// Tests exercise the public input/output and command contracts.
FUNCTION_BLOCK FB_DigitalInput_Test EXTENDS TcUnit.FB_TestSuite

InitialStateClean();
RawSignalPassthroughWithNoDebounce();
InvertFlipsDebouncedValueNotRaw();
RisingEdgePulseOneScan();
FallingEdgePulseOneScan();
DebounceOnBlocksRisingEdgeUntilElapsed();
DebounceOffHoldsSignalHighAfterRawGoesLow();
BadQualityHoldsLastRawValue();
QualityTagSurfacesInStatus();
ClampedQualityReadsAsGood();

METHOD InitialStateClean
VAR
    fb : TcForge.FB_DigitalInput;
END_VAR
TEST('InitialStateClean');

fb(inpQuality := TcForge.E_IO_Quality.GOOD);

AssertFalse(
    Condition := fb.sts.value,
    Message   := 'Fresh instance must read LOW when the physical input is LOW');
AssertFalse(
    Condition := fb.sts.rawValue,
    Message   := 'Fresh instance must report the raw input LOW');
AssertFalse(
    Condition := fb.sts.risingEdge,
    Message   := 'Fresh instance must not emit a spurious rising edge');
AssertFalse(
    Condition := fb.sts.fallingEdge,
    Message   := 'Fresh instance must not emit a spurious falling edge');
AssertFalse(
    Condition := fb.sts.header.faulted,
    Message   := 'Fresh instance must not be faulted');

TEST_FINISHED();
END_METHOD

METHOD RawSignalPassthroughWithNoDebounce
VAR
    fb : TcForge.FB_DigitalInput;
END_VAR
TEST('RawSignalPassthroughWithNoDebounce');

// Default cfg: no debounce, no invert. Raw hardware bit flushes through
// to value in one cycle.
fb.inSignal := TRUE;
fb(inpQuality := TcForge.E_IO_Quality.GOOD);

AssertTrue(
    Condition := fb.sts.rawValue,
    Message   := 'rawValue must echo the hardware bit under GOOD quality');
AssertTrue(
    Condition := fb.sts.value,
    Message   := 'With no debounce and no invert the conditioned value must match the raw bit');

TEST_FINISHED();
END_METHOD

METHOD InvertFlipsDebouncedValueNotRaw
VAR
    fb : TcForge.FB_DigitalInput;
END_VAR
TEST('InvertFlipsDebouncedValueNotRaw');

// Invert must apply to the debounced / published value but the raw
// reading should stay true-to-the-wire so troubleshooters can see what
// the hardware is actually doing.
fb.cfg.invert := TRUE;
fb.inSignal := TRUE;
fb(inpQuality := TcForge.E_IO_Quality.GOOD);

AssertTrue(
    Condition := fb.sts.rawValue,
    Message   := 'rawValue must echo the wire value independent of invert');
AssertFalse(
    Condition := fb.sts.value,
    Message   := 'invert must flip the conditioned value (active-low sensor semantics)');

TEST_FINISHED();
END_METHOD

METHOD RisingEdgePulseOneScan
VAR
    fb : TcForge.FB_DigitalInput;
END_VAR
TEST('RisingEdgePulseOneScan');

fb.inSignal := FALSE;
fb(inpQuality := TcForge.E_IO_Quality.GOOD);

fb.inSignal := TRUE;
fb(inpQuality := TcForge.E_IO_Quality.GOOD);
AssertTrue(
    Condition := fb.sts.risingEdge,
    Message   := 'risingEdge must fire on the cycle the debounced value goes HIGH');

fb(inpQuality := TcForge.E_IO_Quality.GOOD);
AssertFalse(
    Condition := fb.sts.risingEdge,
    Message   := 'risingEdge must clear the very next cycle — edges are one-scan pulses');

TEST_FINISHED();
END_METHOD

METHOD FallingEdgePulseOneScan
VAR
    fb : TcForge.FB_DigitalInput;
END_VAR
TEST('FallingEdgePulseOneScan');

fb.inSignal := TRUE;
fb(inpQuality := TcForge.E_IO_Quality.GOOD);

fb.inSignal := FALSE;
fb(inpQuality := TcForge.E_IO_Quality.GOOD);
AssertTrue(
    Condition := fb.sts.fallingEdge,
    Message   := 'fallingEdge must fire on the cycle the debounced value goes LOW');

fb(inpQuality := TcForge.E_IO_Quality.GOOD);
AssertFalse(
    Condition := fb.sts.fallingEdge,
    Message   := 'fallingEdge must clear the very next cycle');

TEST_FINISHED();
END_METHOD

METHOD DebounceOnBlocksRisingEdgeUntilElapsed
VAR
    fb : TcForge.FB_DigitalInput;
END_VAR
TEST('DebounceOnBlocksRisingEdgeUntilElapsed');

// debounceOn = T#1S — the _tonOn.Q won't fire inside this test frame.
fb.cfg.debounceOn := T#1S;
fb.inSignal := TRUE;
fb(inpQuality := TcForge.E_IO_Quality.GOOD);

AssertTrue(
    Condition := fb.sts.rawValue,
    Message   := 'rawValue must still show the raw bit — debounce gates the conditioned value, not the raw view');
AssertFalse(
    Condition := fb.sts.value,
    Message   := 'debounceOn must hold value LOW until the TON elapses');
AssertFalse(
    Condition := fb.sts.risingEdge,
    Message   := 'No rising edge must be emitted while debounce is pending');

TEST_FINISHED();
END_METHOD

METHOD DebounceOffHoldsSignalHighAfterRawGoesLow
VAR
    fb : TcForge.FB_DigitalInput;
END_VAR
TEST('DebounceOffHoldsSignalHighAfterRawGoesLow');

// debounceOff = T#1S. With debounceOn still 0 we latch the
// debounced signal HIGH immediately, then flip the raw bit LOW and
// expect the TOF to hold the debounced value HIGH.
fb.cfg.debounceOff := T#1S;
fb.inSignal := TRUE;
fb(inpQuality := TcForge.E_IO_Quality.GOOD);
AssertTrue(
    Condition := fb.sts.value,
    Message   := 'Precondition: raw HIGH with zero ON-debounce must latch the debounced value HIGH');

fb.inSignal := FALSE;
fb(inpQuality := TcForge.E_IO_Quality.GOOD);

AssertFalse(
    Condition := fb.sts.rawValue,
    Message   := 'rawValue must immediately mirror the wire going LOW');
AssertTrue(
    Condition := fb.sts.value,
    Message   := 'debounceOff must hold the debounced value HIGH until the TOF expires');
AssertFalse(
    Condition := fb.sts.fallingEdge,
    Message   := 'No falling edge must be emitted while the OFF-debounce is pending');

TEST_FINISHED();
END_METHOD

METHOD BadQualityHoldsLastRawValue
VAR
    fb : TcForge.FB_DigitalInput;
END_VAR
TEST('BadQualityHoldsLastRawValue');

// Latch a known-good HIGH reading.
fb.inSignal := TRUE;
fb(inpQuality := TcForge.E_IO_Quality.GOOD);
AssertTrue(
    Condition := fb.sts.rawValue,
    Message   := 'Precondition: under GOOD quality rawValue mirrors the wire');

// Simulate wire break: the underlying bit flips FALSE but quality is BAD.
// The FB must ignore the glitchy reading and hold the last-known-good raw.
fb.inSignal := FALSE;
fb(inpQuality := TcForge.E_IO_Quality.BAD);

AssertTrue(
    Condition := fb.sts.rawValue,
    Message   := 'BAD quality must freeze rawValue at the last known-good reading');
AssertEquals_USINT(
    Expected := TcForge.E_IO_Quality.BAD,
    Actual   := fb.sts.quality,
    Message  := 'quality must surface the BAD tag so downstream consumers can react');

TEST_FINISHED();
END_METHOD

METHOD QualityTagSurfacesInStatus
VAR
    fb : TcForge.FB_DigitalInput;
END_VAR
TEST('QualityTagSurfacesInStatus');

// UNKNOWN -> BAD -> GOOD must each land in sts.quality unchanged so
// the HMI can display the exact tag the caller supplied.
fb(inpQuality := TcForge.E_IO_Quality.UNKNOWN);
AssertEquals_USINT(
    Expected := TcForge.E_IO_Quality.UNKNOWN,
    Actual   := fb.sts.quality,
    Message  := 'quality must surface UNKNOWN unchanged');

fb(inpQuality := TcForge.E_IO_Quality.BAD);
AssertEquals_USINT(
    Expected := TcForge.E_IO_Quality.BAD,
    Actual   := fb.sts.quality,
    Message  := 'quality must surface BAD unchanged');

fb(inpQuality := TcForge.E_IO_Quality.GOOD);
AssertEquals_USINT(
    Expected := TcForge.E_IO_Quality.GOOD,
    Actual   := fb.sts.quality,
    Message  := 'quality must surface GOOD unchanged');

TEST_FINISHED();
END_METHOD

METHOD ClampedQualityReadsAsGood
VAR
    fb : TcForge.FB_DigitalInput;
END_VAR
TEST('ClampedQualityReadsAsGood');

// The quality gate treats GOOD and CLAMPED as "trust the raw reading".
// CLAMPED is meant for analog signals that hit a scaling limit — for a
// digital input it has to behave the same as GOOD so a wrapper that
// passes CLAMPED through doesn't accidentally freeze the reading.
fb.inSignal := TRUE;
fb(inpQuality := TcForge.E_IO_Quality.CLAMPED);

AssertTrue(
    Condition := fb.sts.rawValue,
    Message   := 'CLAMPED quality must be treated like GOOD for raw readings');
AssertTrue(
    Condition := fb.sts.value,
    Message   := 'CLAMPED quality must not freeze the conditioned value');
AssertEquals_USINT(
    Expected := TcForge.E_IO_Quality.CLAMPED,
    Actual   := fb.sts.quality,
    Message  := 'quality must still surface CLAMPED so consumers know the raw came from a clamped source');

TEST_FINISHED();
END_METHOD

END_FUNCTION_BLOCK

(* stored: Version 1.1.0.1, ProductVersion 3.1.4026.12
   POU FB_DigitalInput_Test: Id {b1c2d3e4-f5a6-7890-abcd-000000000900}, SpecialFunc None
   Method InitialStateClean: Id {b1c2d3e4-f5a6-7890-abcd-000000000901}
   Method RawSignalPassthroughWithNoDebounce: Id {b1c2d3e4-f5a6-7890-abcd-000000000902}
   Method InvertFlipsDebouncedValueNotRaw: Id {b1c2d3e4-f5a6-7890-abcd-000000000903}
   Method RisingEdgePulseOneScan: Id {b1c2d3e4-f5a6-7890-abcd-000000000904}
   Method FallingEdgePulseOneScan: Id {b1c2d3e4-f5a6-7890-abcd-000000000905}
   Method DebounceOnBlocksRisingEdgeUntilElapsed: Id {b1c2d3e4-f5a6-7890-abcd-000000000906}
   Method DebounceOffHoldsSignalHighAfterRawGoesLow: Id {b1c2d3e4-f5a6-7890-abcd-000000000907}
   Method BadQualityHoldsLastRawValue: Id {b1c2d3e4-f5a6-7890-abcd-000000000908}
   Method QualityTagSurfacesInStatus: Id {b1c2d3e4-f5a6-7890-abcd-000000000909}
   Method ClampedQualityReadsAsGood: Id {b1c2d3e4-f5a6-7890-abcd-00000000090a} *)
